(* CoDeSys 2.3.9.47 project: gym_2017_07_09.pr6 *)
(* Libraries: PlcSystemBC.lb6 21.3.01 11:03:02, PlcHelperBC.lb6 7.5.01 11:03:00, TcAdsBC.lb6 5.7.02 11:03:02, standard.lib 5.6.98 11:03:02, TcBABasic.lib 22.7.15 15:46:14, TcPlcUtilitiesBC.lb6 13.5.05 11:19:40 *)

(* Global variable list: main *)
VAR_GLOBAL
	dataDerevo: ARRAY[0..3] OF BYTE;
	dataDerevo_prev :ARRAY[0..3] OF BYTE;

	datafloor1: ARRAY[0..3] OF BYTE;
	datafloor1_prev :ARRAY[0..3] OF BYTE;



	ads_adr_derevo: STRING:='10.0.5.64.1.1';
	ads_adr_3floor: STRING:='10.0.5.63.1.1';
	ads_adr_1floor: STRING:='10.0.5.61.1.1';

	write_ads: ADSWRITE;

	bDarkOutside						AT%MX0.0:BOOL;


	iHour							AT%MB1:	BYTE;
	iMinute							AT%MB3:	BYTE;

	t_out							AT%MB6 :	 REAL;

	eib_gym01 						AT %MX10.0:	 BOOL;
	eib_gym02 						AT %MX10.1:	 BOOL;
	eib_training01 					AT %MX10.2:	 BOOL;
	eib_training02						AT %MX10.3:	 BOOL;
	eib_training03						AT %MX10.4:	 BOOL;
	eib_gym_stairs_bra				AT %MX10.5:	 BOOL;
	eib_pool_hall_spotlight				AT %MX10.6:	 BOOL;
	eib_pool_hall_LED				AT %MX10.7:	 BOOL;

	eib_pool_light 					AT %MX11.0:	 BOOL;
	eib_sphere_ceiling_light 			AT %MX11.1:	 BOOL;
	eib_sphere_light 					AT %MX11.2:	 BOOL;
	eib_gym_cinema_bra 				AT %MX11.3:	 BOOL;
	eib_gym_shower01_light			AT %MX11.4:	 BOOL;
	eib_gym_shower02_light			AT %MX11.5:	 BOOL;
	eib_gym_corridor_light				AT %MX11.6:	 BOOL;
	eib_gym_stairs_light 				AT %MX11.7:	 BOOL;

	eib_gym_WC_light 				AT %MX12.0:	 BOOL;
	eib_training	 					AT %MX12.1:	 BOOL;
	eib_gym		 					AT %MX12.2:	 BOOL;
	eib_outside_bigBulbs		 		AT %MX12.3:	 BOOL;
	eib_outside_pingPongTable		AT %MX12.4:	 BOOL;
	eib_outside_plantsLightning		 	AT %MX12.5:	 BOOL;
	eib_outside_smallBulbs		 	AT %MX12.6:	 BOOL;
	floor1_tambur3_light				AT %MX100.0 :BOOL;
	sw_floor1_tambur3_short			AT %MX100.1 :BOOL;
	sw_floor1_tambur3_long			AT %MX100.2 :BOOL;

END_VAR

(* Global variable list: physical *)
(* @GLOBAL_VARIABLE_LIST := TwinCAT_Import *)
(* @PATH := '' *)
VAR_GLOBAL (* DO NOT CHANGE THIS SHEET MANUALLY! *)
	PlcInVar_0	AT %QB128:	USINT;
	PlcInVar_1	AT %QB129:	USINT;
	PlcInVar_2	AT %QB130:	USINT;
	PlcInVar_3	AT %QB131:	USINT;
	PlcInVar_4	AT %QB132:	USINT;
	PlcInVar_5	AT %QB133:	USINT;
	PlcInVar_6	AT %QB134:	USINT;
	PlcInVar_7	AT %QB135:	USINT;
	PlcInVar_8	AT %QB136:	USINT;
	PlcInVar_9	AT %QB137:	USINT;
	PlcInVar_10	AT %QB138:	USINT;
	PlcInVar_11	AT %QB139:	USINT;
	PlcInVar_12	AT %QB140:	USINT;
	PlcInVar_13	AT %QB141:	USINT;
	PlcInVar_14	AT %QB142:	USINT;
	PlcInVar_15	AT %QB143:	USINT;
	PlcOutVar_0	AT %IB128:	USINT;
	PlcOutVar_1	AT %IB129:	USINT;
	PlcOutVar_2	AT %IB130:	USINT;
	PlcOutVar_3	AT %IB131:	USINT;
	PlcOutVar_4	AT %IB132:	USINT;
	PlcOutVar_5	AT %IB133:	USINT;
	PlcOutVar_6	AT %IB134:	USINT;
	PlcOutVar_7	AT %IB135:	USINT;
	PlcOutVar_8	AT %IB136:	USINT;
	PlcOutVar_9	AT %IB137:	USINT;
	PlcOutVar_10	AT %IB138:	USINT;
	PlcOutVar_11	AT %IB139:	USINT;
	PlcOutVar_12	AT %IB140:	USINT;
	PlcOutVar_13	AT %IB141:	USINT;
	PlcOutVar_14	AT %IB142:	USINT;
	PlcOutVar_15	AT %IB143:	USINT;
	gym01_light				AT %QX0.0:	BOOL; (*K01*)
	training03_light			AT %QX0.1:	BOOL; (*K05*)
	gym02_light				AT %QX0.2:	BOOL; (*K02*)
	gym_stairs_bra_right		AT %QX0.3:	BOOL; (*K06*)
	training01_light			AT %QX0.4:	BOOL; (*K03*)
	gym_stairs_bra_left		AT %QX0.5:	BOOL; (*K07*)
	training02_light			AT %QX0.6:	BOOL; (*K04*)
	pool_hall_spotlight		AT %QX0.7:	BOOL; (*K08*)

	pool_hall_ceiling_LED		AT %QX1.0:	BOOL; (*K09*)
	pool_light				AT %QX1.1:	BOOL; (*K13*)
	sphere_ceiling_light		AT %QX1.2:	BOOL; (*K10*)
	gym01_2_light			AT %QX1.3:	BOOL; (*K14*)
	sphere_light01			AT %QX1.4:	BOOL; (*K11*)
	gym02_2_light			AT %QX1.5:	BOOL; (*K15*)
	gym_cinema_bra			AT %QX1.6:	BOOL; (*K12*)
	training01_2_light			AT %QX1.7:	BOOL; (*K16*)

	training02_2_light			AT %QX2.0:	BOOL; (*K17*)
	gym_shower02_light		AT %QX2.1:	BOOL; (*K21*)
	training03_2_light			AT %QX2.2:	BOOL; (*K18*)
	gym_WC_light			AT %QX2.3:	BOOL; (*K22*)
	gym_shower01_light		AT %QX2.4:	BOOL; (*K19*)
	gym_stairs_light			AT %QX2.5:	BOOL; (*K23*)
	gym_WC_corridor			AT %QX2.6:	BOOL; (*K20*)
	sphere_light02			AT %QX2.7:	BOOL; (*K24*)

	pool_hall_LED			AT %QX3.0:	BOOL; (*K25*)
	outside_smallBulbs		AT %QX3.1:	BOOL;
	gym_cinema_TEMPORARY_light	AT %QX3.2:	BOOL; (*K26*)
	outside_bigBulbs			AT %QX3.3:	BOOL;
	Term_5_KL2408_5_Output	AT %QX3.4:	BOOL;
	outside_plantsLightning	AT %QX3.5:	BOOL;
	Term_5_KL2408_7_Output	AT %QX3.6:	BOOL;
	outside_pingPongTable	AT %QX3.7:	BOOL;

	sw_02_1					AT %IX0.0:	BOOL;
	sw_01_1_2				AT %IX0.1:	BOOL;
	sw_02_2					AT %IX0.2:	BOOL;
	Term_6_KL1408_4_Input	AT %IX0.3:	BOOL;
	sw_03_1					AT %IX0.4:	BOOL;
	sw_01_1_1				AT %IX0.5:	BOOL;
	sw_01_2_1				AT %IX0.6:	BOOL;
	sw_07_1_2				AT %IX0.7:	BOOL;

	sw_07_2_2				AT %IX1.0:	BOOL;
	sw_14_1_1				AT %IX1.1:	BOOL;
	sw_07_2_1				AT %IX1.2:	BOOL;
	sw_14_1_2				AT %IX1.3:	BOOL;
	sw_07_1_1				AT %IX1.4:	BOOL;
	sw_14_2_2				AT %IX1.5:	BOOL;
	Term_7_KL1408_7_Input	AT %IX1.6:	BOOL;
	sw_14_2_1				AT %IX1.7:	BOOL;

	sw_14_3_1				AT %IX2.0:	BOOL;
	sw_09_2_2				AT %IX2.1:	BOOL;
	sw_14_3_2				AT %IX2.2:	BOOL;
	sw_09_3_1				AT %IX2.3:	BOOL;
	sw_09_1_1				AT %IX2.4:	BOOL;
	sw_09_3_2				AT %IX2.5:	BOOL;
	sw_09_2_1				AT %IX2.6:	BOOL;
	sw_09_1_2				AT %IX2.7:	BOOL;

	sw_04_1					AT %IX3.0:	BOOL;
	sw_10_1					AT %IX3.1:	BOOL;
	sw_04_2					AT %IX3.2:	BOOL;
	sw_10_2					AT %IX3.3:	BOOL;
	sw_06_1					AT %IX3.4:	BOOL;
	sw_05_2					AT %IX3.5:	BOOL;
	sw_06_2					AT %IX3.6:	BOOL;
	sw_05_1					AT %IX3.7:	BOOL;

	sw_12_1					AT %IX4.0:	BOOL;
	Term_10_KL1408_2_Input	AT %IX4.1:	BOOL;
	sw_12_2					AT %IX4.2:	BOOL;
	Term_10_KL1408_4_Input	AT %IX4.3:	BOOL;
	Term_10_KL1408_5_Input	AT %IX4.4:	BOOL;
	Term_10_KL1408_6_Input	AT %IX4.5:	BOOL;
	Term_10_KL1408_7_Input	AT %IX4.6:	BOOL;
	Term_10_KL1408_8_Input	AT %IX4.7:	BOOL;
END_VAR

(* @OBJECT_END := TwinCAT_Import *)

(* POU MAIN, ST *)
PROGRAM MAIN
VAR
	i,j:INT;
	write:BOOL;
	heartBeat: TP;
	i1: INT;
	j1: INT;
	write1: BOOL;
	sw_02_1_short_pulse:TP;
	sw_02_1_long_pulse:TP;
	sw_02_2_short_pulse:TP;
	sw_02_2_long_pulse:TP;
	sw_01_2_short_pulse:TP;
	sw_01_2_long_pulse:TP;

	sw_03_1_short_pulse: TP;
	sw_03_1_long_pulse: TP;
END_VAR
heartBeat(IN:= NOT heartBeat.Q, PT:=t#5s);
ADS_Communication;
Light.knx_triggers;
Light;
Light.outsideLight;
(*Counters;*)
write_dataDerevo;
END_PROGRAM
ACTION write_dataDerevo:
	dataDerevo[0].0:= gym01_light ;
	dataDerevo[0].1:= gym02_light;
	dataDerevo[0].2:= training01_light;
	dataDerevo[0].3:= training02_light;
	dataDerevo[0].4:= training03_light;
	dataDerevo[0].5:= gym_stairs_bra_left;
	dataDerevo[0].6:= pool_hall_spotlight;
	dataDerevo[0].7:= pool_hall_LED;

	dataDerevo[1].0:= pool_light;
	dataDerevo[1].1:= sphere_ceiling_light;
	dataDerevo[1].2:= sphere_light01;
	dataDerevo[1].3:= gym_cinema_bra;
	dataDerevo[1].4:= gym_shower01_light;
	dataDerevo[1].5:= gym_shower02_light;
	dataDerevo[1].6:= gym_WC_corridor;
	dataDerevo[1].7:= gym_stairs_light;

	dataDerevo[2].0:= gym_WC_light;
	dataDerevo[2].1:= training03_2_light;
	dataDerevo[2].2:= gym02_2_light;
	dataDerevo[2].3:= outside_bigBulbs;
	dataDerevo[2].4:= outside_pingPongTable;
	dataDerevo[2].5:= outside_plantsLightning;
	dataDerevo[2].6:= outside_smallBulbs;

	sw_02_1_short_pulse(IN:= Light.fb_sw_02_1.bShortClick, pt:=t#500ms);
	sw_02_1_long_pulse(IN:= Light.fb_sw_02_1.bLongClick, pt:=t#500ms);
	sw_02_2_short_pulse(IN:= Light.fb_sw_02_2.bShortClick, pt:=t#500ms);
	sw_02_2_long_pulse(IN:= Light.fb_sw_02_2.bLongClick, pt:=t#500ms);
	sw_01_2_short_pulse(IN:= Light.fb_sw_01_2_1.bShortClick, pt:=t#500ms);
	sw_01_2_long_pulse(IN:= Light.fb_sw_01_2_1.bLongClick, pt:=t#500ms);

	sw_03_1_short_pulse(IN:= Light.fb_sw_03_1.bShortClick, pt:=t#500ms);
	sw_03_1_long_pulse(IN:= Light.fb_sw_03_1.bLongClick, pt:=t#500ms);


	datafloor1[0].0 := sw_02_1_short_pulse.Q;
	datafloor1[0].1 := sw_02_1_long_pulse.Q;
	datafloor1[0].2 := sw_02_2_short_pulse.Q;
	datafloor1[0].3 := sw_02_2_long_pulse.Q;
	datafloor1[0].4 := gym_stairs_bra_left;
	datafloor1[0].5 := sw_01_2_short_pulse.Q;
	datafloor1[0].6 := sw_01_2_long_pulse.Q;
	datafloor1[0].7 := sw_03_1_short_pulse.Q;
	datafloor1[1].0 := sw_03_1_long_pulse.Q;

FOR i:=0 TO (SIZEOF(dataDerevo))-1 DO
	IF dataDerevo[i]<>dataDerevo_prev[i]  THEN
		write:=TRUE;
		EXIT;
	ELSE
		write:=FALSE;
	END_IF
END_FOR


FOR j:=0 TO (SIZEOF(dataDerevo))-1 DO
	dataDerevo_prev[j]:=dataDerevo[j];
END_FOR

FOR i1:=0 TO (SIZEOF(dataFloor1))-1 DO
	IF dataFloor1[i1]<>dataFloor1_prev[i1]  THEN
		write1:=TRUE;
		EXIT;
	ELSE
		write1:=FALSE;
	END_IF
END_FOR


FOR j1:=0 TO (SIZEOF(dataFloor1))-1 DO
	dataFloor1_prev[j1]:=dataFloor1[j1];
END_FOR
END_ACTION

(* POU ADS_Communication, CFC *)
PROGRAM ADS_Communication
VAR
	fb_DerevoADSwrite: ADSWRITE;
	fb_floor1ADSwrite: ADSWRITE;

	counter_error,counter_busy: CTU;
END_VAR
VAR (* helpers for the ST form of the networks *)
	_t21 : DWORD;
	_t23 : DWORD;
	_t42 : BOOL;
	_t50 : DWORD;
	_t52 : DWORD;
	_t56 : BOOL;
END_VAR
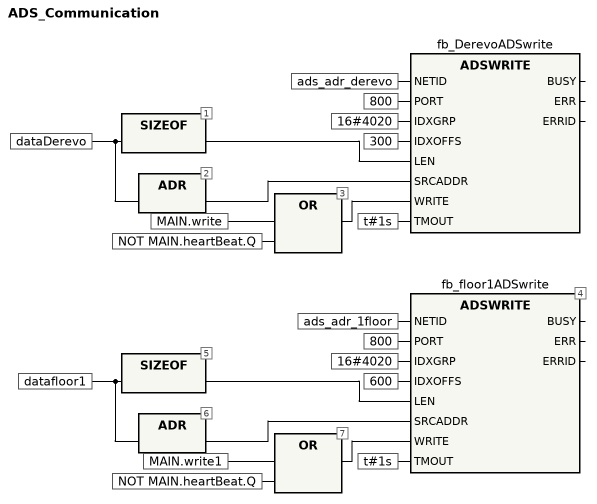
_CFC_ (* Continuous Function Chart, elements in execution order *)
#0 fb_DerevoADSwrite:ADSWRITE(NETID: ads_adr_derevo, PORT: 800, IDXGRP: 16#4020, IDXOFFS: 300, LEN: #1, SRCADDR: #2, WRITE: #3, TMOUT: t#1s)
#1 SIZEOF(dataDerevo)
#2 ADR(dataDerevo)
#3 OR(MAIN.write, NOT MAIN.heartBeat.Q)
#4 fb_floor1ADSwrite:ADSWRITE(NETID: ads_adr_1floor, PORT: 800, IDXGRP: 16#4020, IDXOFFS: 600, LEN: #5, SRCADDR: #6, WRITE: #7, TMOUT: t#1s)
#5 SIZEOF(datafloor1)
#6 ADR(datafloor1)
#7 OR(MAIN.write1, NOT MAIN.heartBeat.Q)
_END_CFC_
(* the same logic as Structured Text *)
fb_DerevoADSwrite(NETID := ads_adr_derevo, PORT := 800, IDXGRP := 16#4020, IDXOFFS := 300, LEN := _t21, SRCADDR := _t23, WRITE := _t42, TMOUT := t#1s);
_t21 := SIZEOF(dataDerevo);
_t23 := ADR(dataDerevo);
_t42 := MAIN.write OR NOT MAIN.heartBeat.Q;
fb_floor1ADSwrite(NETID := ads_adr_1floor, PORT := 800, IDXGRP := 16#4020, IDXOFFS := 600, LEN := _t50, SRCADDR := _t52, WRITE := _t56, TMOUT := t#1s);
_t50 := SIZEOF(datafloor1);
_t52 := ADR(datafloor1);
_t56 := MAIN.write1 OR NOT MAIN.heartBeat.Q;
END_PROGRAM

(* POU Light, CFC *)
PROGRAM Light
VAR
	(*switches*)

	fb_sw_01_1_2	:	FB_ShortLongClick;
	fb_sw_01_1_1	:	FB_ShortLongClick;
	fb_sw_01_2_1	:	FB_ShortLongClick;
	fb_sw_07_1_1	:	FB_ShortLongClick;
	fb_sw_07_2_1	:	FB_ShortLongClick;
	fb_sw_14_1_1	:	FB_ShortLongClick;
	fb_sw_14_1_2	:	FB_ShortLongClick;
	fb_sw_14_2_2	:	FB_ShortLongClick;
	fb_sw_14_2_1	:	FB_ShortLongClick;
	fb_sw_14_3_1	:	FB_ShortLongClick;
	fb_sw_09_2_2	:	FB_ShortLongClick;
	fb_sw_14_3_2	:	FB_ShortLongClick;
	fb_sw_09_3_1	:	FB_ShortLongClick;
	fb_sw_09_1_1	:	FB_ShortLongClick;
	fb_sw_09_3_2	:	FB_ShortLongClick;
	fb_sw_09_2_1	:	FB_ShortLongClick;
	fb_sw_09_1_2	:	FB_ShortLongClick;
	fb_sw_04_1	:	FB_ShortLongClick;
	fb_sw_04_2	:	FB_ShortLongClick;
	fb_sw_06_1	:	FB_ShortLongClick;
	fb_sw_06_2	:	FB_ShortLongClick;

	longPressTimeout	:	TIME := t#500ms;

	(*Lights*)
	fb_gym01_light			: FB_Light;
	fb_gym02_light			: FB_Light;
	fb_training01_light			: FB_Light;
	fb_training02_light			: FB_Light;
	fb_training03_light			: FB_Light;
	fb_gym_stairs_bra			: FB_Light;
	fb_pool_hall_spotlight		: FB_Light;
	fb_pool_hall_LED			: FB_Light;
	fb_pool_light				: FB_Light;
	fb_sphere_ceiling_light		: FB_Light;
	fb_sphere_light			: FB_Light;
	fb_gym_cinema_bra		: FB_Light;
	fb_gym_shower01_light		: FB_Light;
	fb_gym_shower02_light		: FB_Light;
	fb_gym_corridor_light		: FB_Light;
	fb_gym_stairs_light		: FB_Light;
	fb_gym_WC_light			: FB_Light;
	fb_training_light			: FB_Light;
	fb_gym_light				: FB_Light;


	fb_cinema_temporary_light	:FB_Light;

	traning_falling_edge :F_TRIG;
	gym_falling_edge :F_TRIG;


	fb_sw_05_1: FB_ShortLongClick;
	fb_sw_05_2: FB_ShortLongClick;
	fb_training01_2_light: FB_Light;
	fb_gym_01_2_light: FB_Light;
	fb_gym01_2_light: FB_Light;


	rising_edge_eib_gym01 						:	 R_TRIG;
	rising_edge_eib_gym02 						:	 R_trig;
	rising_edge_eib_training01 					:	 R_trig;
	rising_edge_eib_training02						:	 R_trig;
	rising_edge_eib_training03						:	 R_trig;
	rising_edge_eib_gym_stairs_bra				:	 R_trig;
	rising_edge_eib_pool_hall_spotlight				:	 R_trig;
	rising_edge_eib_pool_hall_LED				:	 R_trig;

	rising_edge_eib_pool_light 					:	 R_trig;
	rising_edge_eib_sphere_ceiling_light 			:	 R_trig;
	rising_edge_eib_sphere_light 					:	 R_trig;
	rising_edge_eib_gym_cinema_bra 				:	 R_trig;
	rising_edge_eib_gym_shower01_light			:	 R_trig;
	rising_edge_eib_gym_shower02_light			:	 R_trig;
	rising_edge_eib_gym_corridor_light				:	 R_trig;
	rising_edge_eib_gym_stairs_light 				:	 R_trig;

	rising_edge_eib_gym_WC_light 				:	 R_trig;
	rising_edge_eib_training	 					:	 R_trig;
	rising_edge_eib_gym		 					:	 R_TRIG;

	falling_edge_eib_gym01 						:	 F_TRIG;
	falling_edge_eib_gym02 						:	 F_TRIG;
	falling_edge_eib_training01 					:	 F_TRIG;
	falling_edge_eib_training02						:	 F_TRIG;
	falling_edge_eib_training03						:	 F_TRIG;
	falling_edge_eib_gym_stairs_bra				:	 F_TRIG;
	falling_edge_eib_pool_hall_spotlight				:	 F_TRIG;
	falling_edge_eib_pool_hall_LED				:	 F_TRIG;

	falling_edge_eib_pool_light 					:	 F_TRIG;
	falling_edge_eib_sphere_ceiling_light 			:	 F_TRIG;
	falling_edge_eib_sphere_light 					:	 F_TRIG;
	falling_edge_eib_gym_cinema_bra 				:	 F_TRIG;
	falling_edge_eib_gym_shower01_light			:	 F_TRIG;
	falling_edge_eib_gym_shower02_light			:	 F_TRIG;
	falling_edge_eib_gym_corridor_light				:	 F_TRIG;
	falling_edge_eib_gym_stairs_light 				:	 F_TRIG;

	falling_edge_eib_gym_WC_light 				:	 F_TRIG;
	falling_edge_eib_training	 					:	 F_TRIG;
	falling_edge_eib_gym		 					:	 F_TRIG;

	(*timers*)
	fb_OutsideLightTimer	:TP;

	fb_pool_hall_all: FB_Light;
	pool_all_falling_edge: F_TRIG;
	pool_all_rising_edge: R_TRIG;
	pool_hall_all_rising_edge: R_TRIG;
	pool_hall_all_falling_edge: F_TRIG;
	traning_reserved_falling_edge: F_TRIG;
	fb_sw_07_1_2: FB_ShortLongClick;
	fb_sw_07_2_2: FB_ShortLongClick;
	fb_sw_02_1: FB_ShortLongClick;
	fb_sw_02_2: FB_ShortLongClick;
	fb_sw_03_1: FB_ShortLongClick;
	darkOutside_rising_edge:R_TRIG;

	darkness_correction_time_hour:INT := 20;

END_VAR
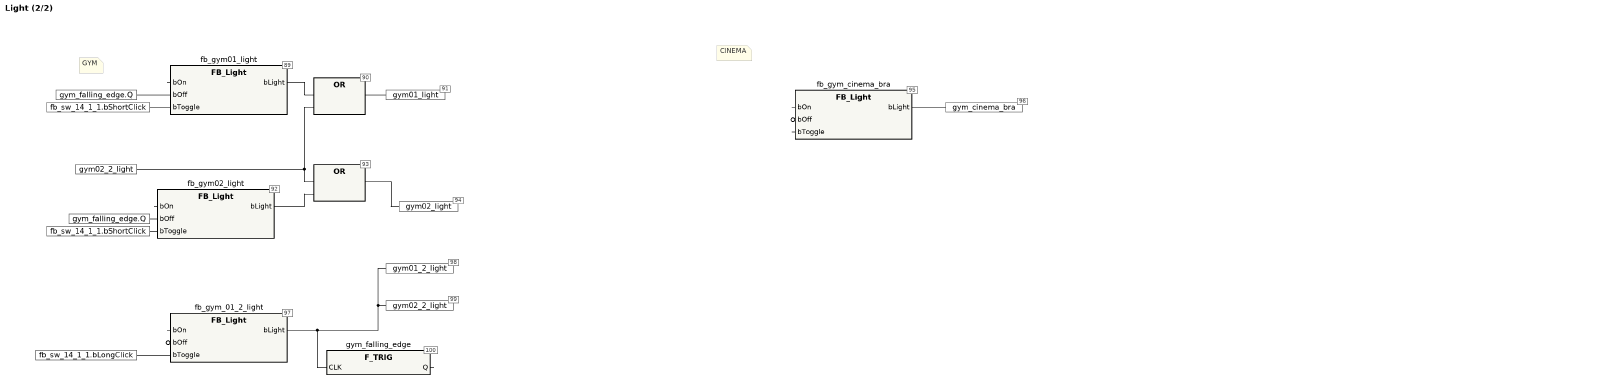
_CFC_ (* Continuous Function Chart, elements in execution order *)
(* GYM *)
(* CINEMA *)
(* SHOWER *)
(* SPHERE *)
(* POOL HALL *)
(* TRAINING *)
(* STAIRS *)
#0 fb_sw_01_1_1:FB_ShortLongClick(bSwitch: sw_01_1_1, tSwitchTime: longPressTimeout)
#1 fb_sw_04_1:FB_ShortLongClick(bSwitch: sw_04_1, tSwitchTime: longPressTimeout)
#2 fb_sw_07_1_1:FB_ShortLongClick(bSwitch: sw_07_1_1, tSwitchTime: longPressTimeout)
#3 fb_sw_09_1_1:FB_ShortLongClick(bSwitch: sw_09_1_1, tSwitchTime: longPressTimeout)
#4 fb_sw_14_1_1:FB_ShortLongClick(bSwitch: sw_14_1_1, tSwitchTime: longPressTimeout)
#5 fb_sw_01_1_2:FB_ShortLongClick(bSwitch: sw_01_1_2, tSwitchTime: longPressTimeout)
#6 fb_sw_04_2:FB_ShortLongClick(bSwitch: sw_04_2, tSwitchTime: longPressTimeout)
#7 fb_sw_07_1_2:FB_ShortLongClick(bSwitch: sw_07_1_2, tSwitchTime: longPressTimeout)
#8 fb_sw_09_1_2:FB_ShortLongClick(bSwitch: sw_09_1_2, tSwitchTime: longPressTimeout)
#9 fb_sw_14_1_2:FB_ShortLongClick(bSwitch: sw_14_1_2, tSwitchTime: longPressTimeout)
#10 fb_sw_05_1:FB_ShortLongClick(bSwitch: sw_05_1, tSwitchTime: longPressTimeout)
#11 fb_sw_07_2_1:FB_ShortLongClick(bSwitch: sw_07_2_1, tSwitchTime: longPressTimeout)
#12 fb_sw_09_2_1:FB_ShortLongClick(bSwitch: sw_09_2_1, tSwitchTime: longPressTimeout)
#13 fb_sw_14_2_1:FB_ShortLongClick(bSwitch: sw_14_2_1, tSwitchTime: longPressTimeout)
#14 fb_sw_01_2_1:FB_ShortLongClick(bSwitch: sw_01_2_1, tSwitchTime: longPressTimeout)
#15 fb_sw_05_2:FB_ShortLongClick(bSwitch: sw_05_2, tSwitchTime: longPressTimeout)
#16 fb_sw_07_2_2:FB_ShortLongClick(bSwitch: sw_07_2_2, tSwitchTime: longPressTimeout)
#17 fb_sw_09_2_2:FB_ShortLongClick(bSwitch: sw_09_2_2, tSwitchTime: longPressTimeout)
#18 fb_sw_14_2_2:FB_ShortLongClick(bSwitch: sw_14_2_2, tSwitchTime: longPressTimeout)
#19 fb_sw_06_1:FB_ShortLongClick(bSwitch: sw_06_1, tSwitchTime: longPressTimeout)
#20 fb_sw_02_1:FB_ShortLongClick(bSwitch: sw_02_1, tSwitchTime: longPressTimeout)
#21 fb_sw_09_3_1:FB_ShortLongClick(bSwitch: sw_09_3_1, tSwitchTime: longPressTimeout)
#22 fb_sw_14_3_1:FB_ShortLongClick(bSwitch: sw_14_3_1, tSwitchTime: longPressTimeout)
#23 fb_sw_06_2:FB_ShortLongClick(bSwitch: sw_06_2, tSwitchTime: longPressTimeout)
#24 fb_sw_09_3_2:FB_ShortLongClick(bSwitch: sw_09_3_2, tSwitchTime: longPressTimeout)
#25 fb_sw_14_3_2:FB_ShortLongClick(bSwitch: sw_14_3_2, tSwitchTime: longPressTimeout)
#26 fb_sw_02_2:FB_ShortLongClick(bSwitch: sw_02_2, tSwitchTime: longPressTimeout)
#27 fb_sw_03_1:FB_ShortLongClick(bSwitch: sw_03_1, tSwitchTime: longPressTimeout)
#28 fb_training01_2_light:FB_Light(bOn: -, bOff: traning_falling_edge.Q, bToggle: fb_sw_01_1_1.bLongClick)
#29 OR(fb_sw_01_1_2.bLongClick, fb_sw_05_2.bLongClick, fb_sw_09_3_2.bLongClick)
#30 fb_training_light:FB_Light(bOn: -, bOff: -, bToggle: #29)
#31 training02_2_light <= #30.bLight
#32 training03_2_light <= #30.bLight
#33 OR(#28.bLight, #30.bLight)
#34 training01_2_light <= #33
#35 traning_falling_edge:F_TRIG(CLK: #30.bLight)
#36 OR(traning_falling_edge.Q, traning_reserved_falling_edge.Q)
#37 fb_training01_light:FB_Light(bOn: -, bOff: #36, bToggle: fb_sw_01_1_1.bShortClick)
#38 OR(#37.bLight, training01_2_light, training02_light)
#39 training01_light <= #38
#40 OR(fb_sw_01_1_2.bShortClick, fb_sw_09_3_2.bShortClick, fb_sw_05_2.bShortClick)
#41 fb_training02_light:FB_Light(bOn: -, bOff: traning_falling_edge.Q, bToggle: #40)
#42 traning_reserved_falling_edge:F_TRIG(CLK: #41.bLight)
#43 OR(#41.bLight, training02_2_light)
#44 training02_light <= #43
#45 fb_training03_light:FB_Light(bOn: -, bOff: traning_falling_edge.Q, bToggle: #40)
#46 OR(#45.bLight, training03_2_light)
#47 training03_light <= #46
#48 OR(fb_sw_09_2_1.bShortClick, fb_sw_14_2_2.bShortClick)
#49 AND(fb_pool_hall_LED.bLight, fb_pool_hall_spotlight.bLight, pool_hall_all_falling_edge.Q)
#50 fb_pool_hall_LED:FB_Light(bOn: pool_hall_all_rising_edge.Q, bOff: #49, bToggle: #48)
#51 pool_hall_ceiling_LED <= #50.bLight
#52 pool_hall_LED <= #50.bLight
#53 OR(fb_sw_09_2_2.bShortClick, fb_sw_14_2_1.bShortClick)
#54 fb_pool_hall_spotlight:FB_Light(bOn: pool_hall_all_rising_edge.Q, bOff: #49, bToggle: #53)
#55 pool_hall_spotlight <= #54.bLight
#56 AND(#50.bLight, #54.bLight)
#57 pool_all_falling_edge:F_TRIG(CLK: #56)
#58 pool_all_rising_edge:R_TRIG(CLK: #56)
#59 OR(fb_sw_09_2_1.bLongClick, fb_sw_14_2_2.bLongClick, fb_sw_09_2_2.bLongClick, fb_sw_14_2_1.bLongClick)
#60 fb_pool_hall_all:FB_Light(bOn: pool_all_rising_edge.Q, bOff: pool_all_falling_edge.Q, bToggle: #59)
#61 pool_hall_all_falling_edge:F_TRIG(CLK: #60.bLight)
#62 pool_hall_all_rising_edge:R_TRIG(CLK: #60.bLight)
#63 OR(fb_sw_09_1_2.bLongClick, fb_sw_14_3_1.bLongClick)
#64 fb_pool_light:FB_Light(bOn: -, bOff: -, bToggle: #63)
#65 pool_light <= #102
#66 AND(fb_sw_05_1.bLongClick, fb_sphere_light.bLight, fb_sphere_ceiling_light.bLight)
#67 fb_sphere_light:FB_Light(bOn: -, bOff: #66, bToggle: fb_sw_05_1.bLongClick)
#68 sphere_light01 <= #67.bLight
#69 sphere_light02 <= #67.bLight
#70 fb_sphere_ceiling_light:FB_Light(bOn: -, bOff: #66, bToggle: fb_sw_05_1.bShortClick)
#71 OR(#67.bLight, #70.bLight)
#72 sphere_ceiling_light <= #71
#73 fb_gym_shower01_light:FB_Light(bOn: -, bOff: -, bToggle: fb_sw_07_1_2.bShortClick)
#74 gym_shower01_light <= #73.bLight
#75 XOR(floor1_tambur3_light, gym_stairs_bra_left)
#76 AND(#75, #101)
#77 OR(fb_sw_02_2.bShortClick, fb_sw_02_2.bLongClick, fb_sw_02_1.bLongClick, #76, fb_sw_01_2_1.bLongClick, fb_sw_01_2_1.bShortClick)
#78 fb_gym_stairs_bra:FB_Light(bOn: -, bOff: -, bToggle: #77)
#79 gym_stairs_bra_left <= #78.bLight
#80 gym_stairs_bra_right <= #78.bLight
#81 fb_gym_shower02_light:FB_Light(bOn: -, bOff: -, bToggle: fb_sw_07_1_1.bShortClick)
#82 gym_shower02_light <= #81.bLight
#83 fb_gym_stairs_light:FB_Light(bOn: -, bOff: -, bToggle: -)
#84 gym_stairs_light <= #83.bLight
#85 fb_gym_WC_light:FB_Light(bOn: -, bOff: -, bToggle: fb_sw_07_2_1.bShortClick)
#86 gym_WC_light <= #85.bLight
#87 fb_gym_corridor_light:FB_Light(bOn: -, bOff: -, bToggle: fb_sw_07_2_2.bShortClick)
#88 gym_WC_corridor <= #87.bLight
#89 fb_gym01_light:FB_Light(bOn: -, bOff: gym_falling_edge.Q, bToggle: fb_sw_14_1_1.bShortClick)
#90 OR(#89.bLight, gym02_2_light)
#91 gym01_light <= #90
#92 fb_gym02_light:FB_Light(bOn: -, bOff: gym_falling_edge.Q, bToggle: fb_sw_14_1_1.bShortClick)
#93 OR(gym02_2_light, #92.bLight)
#94 gym02_light <= #93
#95 fb_gym_cinema_bra:FB_Light(bOn: -, bOff: -, bToggle: -)
#96 gym_cinema_bra <= #95.bLight
#97 fb_gym_01_2_light:FB_Light(bOn: -, bOff: -, bToggle: fb_sw_14_1_1.bLongClick)
#98 gym01_2_light <= #97.bLight
#99 gym02_2_light <= #97.bLight
#100 gym_falling_edge:F_TRIG(CLK: #97.bLight)
#101 OR(sw_floor1_tambur3_short, sw_floor1_tambur3_long)
unconnected input fb_sw_09_2_1.bLongClick
unconnected input fb_sw_14_2_2.bLongClick
#102 OR(sw_09_1_2, sw_14_3_1)
_END_CFC_
END_PROGRAM
ACTION knx_triggers:
	rising_edge_eib_gym01 						(CLK:= eib_gym01);
	rising_edge_eib_gym02 						(CLK:= eib_gym02);
	rising_edge_eib_training01 					(CLK:= eib_training01);
	rising_edge_eib_training02						(CLK:=eib_training02 );
	rising_edge_eib_training03						(CLK:= eib_training03);
	rising_edge_eib_gym_stairs_bra				(CLK:= eib_gym_stairs_bra);
	rising_edge_eib_pool_hall_spotlight				(CLK:=eib_pool_hall_spotlight );
	rising_edge_eib_pool_hall_LED				(CLK:= eib_pool_hall_LED);

	rising_edge_eib_pool_light 					(CLK:= eib_pool_light);
	rising_edge_eib_sphere_ceiling_light 			(CLK:= eib_sphere_ceiling_light);
	rising_edge_eib_sphere_light 					(CLK:= eib_sphere_light);
	rising_edge_eib_gym_cinema_bra 				(CLK:= eib_gym_cinema_bra);
	rising_edge_eib_gym_shower01_light			(CLK:= eib_gym_shower01_light);
	rising_edge_eib_gym_shower02_light			(CLK:= eib_gym_shower02_light);
	rising_edge_eib_gym_corridor_light				(CLK:= eib_gym_corridor_light);
	rising_edge_eib_gym_stairs_light 				(CLK:= eib_gym_stairs_light);

	rising_edge_eib_gym_WC_light 				(CLK:= eib_gym_WC_light);
	rising_edge_eib_training	 					(CLK:= eib_training);
	rising_edge_eib_gym		 					(CLK:= eib_gym);

	falling_edge_eib_gym01 						(CLK:= eib_gym01);
	falling_edge_eib_gym02 						(CLK:= eib_gym02);
	falling_edge_eib_training01 					(CLK:= eib_training01);
	falling_edge_eib_training02						(CLK:=eib_training02 );
	falling_edge_eib_training03						(CLK:= eib_training03);
	falling_edge_eib_gym_stairs_bra				(CLK:= eib_gym_stairs_bra);
	falling_edge_eib_pool_hall_spotlight				(CLK:=eib_pool_hall_spotlight );
	falling_edge_eib_pool_hall_LED				(CLK:= eib_pool_hall_LED);

	falling_edge_eib_pool_light 					(CLK:= eib_pool_light);
	falling_edge_eib_sphere_ceiling_light 			(CLK:= eib_sphere_ceiling_light);
	falling_edge_eib_sphere_light 					(CLK:= eib_sphere_light);
	falling_edge_eib_gym_cinema_bra 				(CLK:= eib_gym_cinema_bra);
	falling_edge_eib_gym_shower01_light			(CLK:= eib_gym_shower01_light);
	falling_edge_eib_gym_shower02_light			(CLK:= eib_gym_shower02_light);
	falling_edge_eib_gym_corridor_light				(CLK:= eib_gym_corridor_light);
	falling_edge_eib_gym_stairs_light 				(CLK:= eib_gym_stairs_light);

	falling_edge_eib_gym_WC_light 				(CLK:= eib_gym_WC_light);
	falling_edge_eib_training	 					(CLK:= eib_training);
	falling_edge_eib_gym		 					(CLK:= eib_gym);
END_ACTION
ACTION outsideLight:
darkOutside_rising_edge(CLK:=bDarkOutside);
IF  bdarkOutside AND (iHour <1 OR iHour>=20) AND iminute=59 THEN
	outside_bigBulbs := TRUE;
	eib_outside_bigBulbs:=TRUE;
	outside_plantsLightning:=TRUE;
	eib_outside_plantsLightning := TRUE;
	outside_smallBulbs := TRUE;
	eib_outside_smallBulbs:= TRUE;
	outside_pingPongTable := FALSE;



ELSE
	outside_bigBulbs := eib_outside_bigBulbs;
	outside_plantsLightning:= eib_outside_plantsLightning;
	outside_smallBulbs := eib_outside_smallBulbs;
	outside_pingPongTable:=eib_outside_pingPongTable;

	IF iHour=2 AND iMinute>=1 AND iMinute<=2 THEN
		outside_bigBulbs := FALSE;
		outside_plantsLightning:=FALSE;
		outside_smallBulbs := FALSE;
		outside_pingPongTable := FALSE;
	END_IF

END_IF;
END_ACTION

(* POU Counters, ST *)
PROGRAM Counters
VAR

	counter_6_KL1408_1_Input : CTU;

	counter_6_KL1408_3_Input	:	CTU;
	counter_6_KL1408_4_Input	:	CTU;
	counter_6_KL1408_5_Input	:	CTU;
	counter_6_KL1408_6_Input	:	CTU;

	counter_6_KL1408_8_Input	:	CTU;
	counter_7_KL1408_1_Input	:	CTU;
	counter_7_KL1408_2_Input	:	CTU;
	counter_7_KL1408_3_Input	:	CTU;
	counter_7_KL1408_4_Input	:	CTU;
	counter_7_KL1408_5_Input	:	CTU;
	counter_7_KL1408_6_Input	:	CTU;
	counter_7_KL1408_7_Input	:	CTU;
	counter_7_KL1408_8_Input	:	CTU;
	counter_8_KL1408_1_Input	:	CTU;
	counter_8_KL1408_2_Input	:	CTU;
	counter_8_KL1408_3_Input	:	CTU;
	counter_8_KL1408_4_Input	:	CTU;
	counter_8_KL1408_5_Input	:	CTU;
	counter_8_KL1408_6_Input	:	CTU;
	counter_8_KL1408_7_Input	:	CTU;
	counter_8_KL1408_8_Input	:	CTU;
	counter_9_KL1408_1_Input	:	CTU;
	counter_9_KL1408_2_Input	:	CTU;
	counter_9_KL1408_3_Input	:	CTU;
	counter_9_KL1408_4_Input	:	CTU;
	counter_9_KL1408_5_Input	:	CTU;
	counter_9_KL1408_6_Input	:	CTU;
	counter_9_KL1408_7_Input	:	CTU;
	counter_9_KL1408_8_Input	:	CTU;
	counter_10_KL1408_1_Input	:	CTU;
	counter_10_KL1408_2_Input	:	CTU;
	counter_10_KL1408_3_Input	:	CTU;
	counter_10_KL1408_4_Input	:	CTU;
	counter_10_KL1408_5_Input	:	CTU;
	counter_10_KL1408_6_Input	:	CTU;
	counter_10_KL1408_7_Input	:	CTU;
	counter_10_KL1408_8_Input	:	CTU;

	sw01 : INT;
	sw02 : INT;
	sw03 : INT;
	sw04 : INT;
	sw05 : INT;
	sw06 : INT;
	sw07 : INT;
	sw08 : INT;
	sw09 : INT;
	sw10 : INT;
	sw11 : INT;
	sw12 : INT;
	sw13 : INT;
	sw14 : INT;
	sw15 : INT;
	sw16 : INT;
	sw17 : INT;
	sw18 : INT;
	sw19 : INT;
	sw20 : INT;
	sw21 : INT;
	sw22 : INT;
	sw23 : INT;
	sw24 : INT;
	sw25 : INT;
	sw26 : INT;
	sw27 : INT;
	sw28 : INT;
	sw29 : INT;
	sw30 : INT;
	sw31 : INT;
	sw32 : INT;
	sw33 : INT;
	sw34 : INT;
	sw35 : INT;
	sw36 : INT;
	sw37 : INT;
	sw38 : INT;
	sw39 : INT;


END_VAR
	counter_6_KL1408_1_Input(CU:= Term_6_KL1408_1_Input, CV=>sw01);

	counter_6_KL1408_3_Input(CU:= Term_6_KL1408_3_Input, CV=>sw02);
	counter_6_KL1408_4_Input(CU:= Term_6_KL1408_4_Input, CV=>sw03);
	counter_6_KL1408_5_Input(CU:= Term_6_KL1408_5_Input, CV=>sw04);





	counter_7_KL1408_3_Input(CU:= Term_7_KL1408_3_Input, CV=>sw09);

	counter_7_KL1408_5_Input(CU:= Term_7_KL1408_5_Input, CV=>sw11);

	counter_7_KL1408_7_Input(CU:= Term_7_KL1408_7_Input, CV=>sw13);












	counter_9_KL1408_2_Input(CU:= Term_9_KL1408_2_Input, CV=>sw24);

	counter_9_KL1408_4_Input(CU:= Term_9_KL1408_4_Input, CV=>sw26);

	counter_9_KL1408_6_Input(CU:= Term_9_KL1408_6_Input, CV=>sw28);

	counter_9_KL1408_8_Input(CU:= Term_9_KL1408_8_Input, CV=>sw30);

	counter_10_KL1408_1_Input(CU:= Term_10_KL1408_1_Input, CV=>sw31);
	counter_10_KL1408_2_Input(CU:= Term_10_KL1408_2_Input, CV=>sw32);
	counter_10_KL1408_3_Input(CU:= Term_10_KL1408_3_Input, CV=>sw33);
	counter_10_KL1408_4_Input(CU:= Term_10_KL1408_4_Input, CV=>sw34);
	counter_10_KL1408_5_Input(CU:= Term_10_KL1408_5_Input, CV=>sw35);
	counter_10_KL1408_6_Input(CU:= Term_10_KL1408_6_Input, CV=>sw36);
	counter_10_KL1408_7_Input(CU:= Term_10_KL1408_7_Input, CV=>sw37);
	counter_10_KL1408_8_Input(CU:= Term_10_KL1408_8_Input, CV=>sw38);
END_PROGRAM
